// TIA Portal V18 export
// export: Created 2026-01-09T11:32:01.5615345Z, ExportSetting WithDefaults, DisplayName Totally Integrated Automation Portal, DisplayVersion V18 Update 5, DisplayName TIA Portal Openness, DisplayVersion V18 Update 5, DisplayName TIA Portal Teamcenter Gateway, DisplayVersion V18, DisplayName TIA Portal Version Control Interface, DisplayVersion V18, DisplayName SINAMICS Startdrive Advanced, DisplayVersion V18 SP2 Update 1, DisplayName SINAMICS Startdrive G110M, G120, G120C, G120D, G120P, G115D, DisplayVersion V18 SP2 Update 1, DisplayName SINAMICS Startdrive G130, G150, S120, S150, SINAMICS MV, S210, G220, S200, DisplayVersion V18 SP2 Update 1, DisplayName STEP 7 Professional, DisplayVersion V18 Update 5, DisplayName STEP 7 Safety, DisplayVersion V18, DisplayName WinCC Professional, DisplayVersion V18 Update 5
TagTable "Com"
  Sys_COM_FlashTime100mS : Bool  (PLC tag Sys.COM.FlashTime100mS, CPU S71500-2PN_TP700, 100 ms)
  Sys_COM_FlashTime200mS : Bool  (PLC tag Sys.COM.FlashTime200mS, CPU S71500-2PN_TP700, 100 ms)
    on ChangeValue: VBCom(Index := 4); LoadCurrentProduct(ProductType := Sys_VersionManagement_StationID)
  Sys_COM_FlashTime500mS : Bool  (PLC tag Sys.COM.FlashTime500mS, CPU S71500-2PN_TP700, 100 ms)
  Sys_COM_FlashTime1S : Bool  (PLC tag Sys.COM.FlashTime1S, CPU S71500-2PN_TP700, 100 ms)
  Sys_COM_FlashTime2S : Bool  (PLC tag Sys.COM.FlashTime2S, CPU S71500-2PN_TP700, 100 ms)
  Sys_COM_AlwaysON : Bool  (PLC tag Sys.COM.AlwaysON, %DB3000.DBX0.1, CPU S71500-2PN_TP700, 1 s)
  Sys_DateTime_Set : Date_And_Time  (PLC tag Sys.DateTime.Set, %DB3000.DBX10.0, CPU S71500-2PN_TP700, 1 s, start 01/01/1999 12:00:00)
  Sys_DateTime_Read : Date_And_Time  (PLC tag Sys.DateTime.Read, %DB3000.DBX18.0, CPU S71500-2PN_TP700, 1 s, start 01/01/1999 12:00:00)
  Sys_DateTime_Trigger : Bool  (PLC tag Sys.DateTime.Trigger, %DB3000.DBX26.0, CPU S71500-2PN_TP700, 1 s)   // Set
  SysComFlashTime100mS : Bool  (PLC tag Sys.COM.FlashTime100mS, CPU S71500-2PN_TP700, 100 ms)
  SysComFlashTime200mS : Bool  (PLC tag Sys.COM.FlashTime200mS, CPU S71500-2PN_TP700, 100 ms)
  SysComFlashTime500mS : Bool  (PLC tag Sys.COM.FlashTime500mS, CPU S71500-2PN_TP700, 100 ms)
  SysComFlashTime1S : Bool  (PLC tag Sys.COM.FlashTime1S, CPU S71500-2PN_TP700, 100 ms)
  SysComFlashTime2S : Bool  (PLC tag Sys.COM.FlashTime2S, CPU S71500-2PN_TP700, 100 ms)
  SysComAlwaysON : Bool  (PLC tag Sys.COM.AlwaysON, %DB3000.DBX0.1, CPU S71500-2PN_TP700, 1 s)
  SysDateTimeSet : Date_And_Time  (PLC tag Sys.DateTime.Set, %DB3000.DBX10.0, CPU S71500-2PN_TP700, 1 s, start 01/01/1999 12:00:00)
  SysDateTimeRead : Date_And_Time  (PLC tag Sys.DateTime.Read, %DB3000.DBX18.0, CPU S71500-2PN_TP700, 1 s, start 01/01/1999 12:00:00)
  SysDateTimeTrigger : Bool  (PLC tag Sys.DateTime.Trigger, %DB3000.DBX26.0, CPU S71500-2PN_TP700, 1 s)
